# EPICS substitutions: iocBoot/ioc13bma_linux/MeasCompAliases.substitutions
file "$(CARS)/db/analog_out_alias.template"
{
pattern
{      REC,              ALIAS,           EGUL,  DRVL,  LOPR,  EGUF,  DRVH,  HOPR, PREC,       DESC}
{13BMA:E1608:Ao1,  13BMA:MonoPiezoPitch,  -10,   -10,    -10,   10,    10,    10,    3,   "Monochromator piezo pitch"}
}
